(****************************************************************************************)
(*							Beckhoff Automation Poland									*)
(*							L_TBConvWordToBits v1.0										*)
(*									29.02.2007											*)
(*	This FB returns the 16 corresponding bit values for an input value of type ” word”	*)
(*______________________________________________________________________________________*)
FUNCTION_BLOCK L_TBConvWordToBits
VAR_INPUT
	wInput:WORD;
END_VAR
VAR_OUTPUT
	bBit0: BOOL;
	bBit1: BOOL;
	bBit2: BOOL;
	bBit3: BOOL;
	bBit4: BOOL;
	bBit5: BOOL;
	bBit6: BOOL;
	bBit7: BOOL;
	bBit8: BOOL;
	bBit9: BOOL;
	bBit10: BOOL;
	bBit11: BOOL;
	bBit12: BOOL;
	bBit13: BOOL;
	bBit14: BOOL;
	bBit15: BOOL;
END_VAR
VAR
END_VAR

bBit0:=wInput.0;
bBit1:=wInput.1;
bBit2:=wInput.2;
bBit3:=wInput.3;
bBit4:=wInput.4;
bBit5:=wInput.5;
bBit6:=wInput.6;
bBit7:=wInput.7;
bBit8:=wInput.8;
bBit9:=wInput.9;
bBit10:=wInput.10;
bBit11:=wInput.11;
bBit12:=wInput.12;
bBit13:=wInput.13;
bBit14:=wInput.14;
bBit15:=wInput.15;

END_FUNCTION_BLOCK

(* stored: Version 1.1.0.1, ProductVersion 3.1.4026.13, FileIdentifier 26800edd48d1477d1476804a84f674382454e2b6, FileSignature 199fa064c0fac833ba8aa31512a2430d17e0ecfe471ef012b27a9ae8a15be5f436cc53721ea508137db70a39898d34008648c48b0a515c6c6505cbbaacabe67e02c17caaa0b7b3a849a66f3da22e96642481eb3227b7e586abd782536acfb9f1f36a7c59722658c985caf922c50301d701b99dfe92c6dbd37f4d7ed5510c68318aefc5be9429d07553f27a1ec3e3136aa230e43ff472f86c2ed865c2d6c416bc3322395ef66fb72eaf9ab50d1d16cd82174d97126df4b830e45ceb7165c3c4654cf78f9035f2e497bb1c37d7950d8dca81f173dedb8cb1133240690f93321205fed7ba6cbd4d6797b2df01b6900b24de91558536e6991882bc42d3c38c2e2e4b
   POU L_TBConvWordToBits: Id {7d26c52e-8d4e-4bcf-b775-741690c99f76}, SpecialFunc None *)
